Staubli VAL3: Control_Mess.pgx

public program Control_Mess(string x_sMess, string x_sLable)
begin

  setTextMode(0)
gotoxy(0,1)
put(x_sMess)
  gotoxy(0,2)
put(x_sLable)

end
